PROGRAM PRG_LVCP1_PowerMeasurement
VAR
	// Enerji Yönetimi
	fbEL3453	: FB_EL3453;	
	stEL3453	: stEL3453;
END_VAR


	fbEL3453(pOut := ADR(stEL3453));

END_PROGRAM

(* stored: Version 1.1.0.1, ProductVersion 3.1.4024.15
   POU PRG_LVCP1_PowerMeasurement: Id {1ea839ba-2e9f-4299-a6f2-957244b1f91c}, SpecialFunc None *)
